# EPICS autosave request: iocBoot/iocTestBusyAsyn/auto_settings.req
$(P)busy1
$(P)busy2
$(P)busy3
$(P)busy4
